# B&R Automation Studio project Prog_2
Automation Studio 4.5.2.102

## Configuration Config1

### Task classes (Cpu.sw)
```
Cyclic#1:
  Program <- Program.prg
Binaries: udbdef, TCData, ashwd, User, asfw, arconfig, sysconf, Role, ashwac, iomap, OpcUaMap
```

### Hardware
```
4PP065_0571_P74 : 4PP065.0571-P74 v1.1.2.0
  Connector IF5:
    ActivateDevice = 1
  ConfigurationID = Prog_2_Config1
  Simulation = 1
  ActivateOpcUa = 1
  OpcUa_SamplingTimer_Default = 1
  OpcUaInformationModels_PV_Version = 1
```

## Logical view

### Global.var
```iecst
VAR
	VP_At_Entry : BOOL;
	VP_At_Exit : BOOL;
	VP_Buffer_Conveyor : BOOL;
	VP_Entry_Conveyor : BOOL;
	VP_Item_Ready : BOOL;
	VP_Start_Button : BOOL;
	VP_Stop_Button : BOOL;
	VP_Dose_Button : BOOL;
END_VAR
```

### Program Logical/Program

#### Variables.var
```iecst
VAR
	RUN : BOOL;
	ENTRY_RUN : BOOL;
	DOSE : BOOL;
	RUN_TIME : UINT;
END_VAR
```

#### Main.c
```c
#include <bur/plctypes.h>

#ifdef _DEFAULT_INCLUDES
	#include <AsDefault.h>
#endif

void _INIT ProgramInit(void)
{

}

void _CYCLIC ProgramCyclic(void)
{
	if (VP_Start_Button) RUN = 1;
	if (!VP_Stop_Button) RUN = 0;

	if (RUN) {
		VP_Buffer_Conveyor = 1;

		if (!VP_Item_Ready) ENTRY_RUN = 1;
		if (VP_Dose_Button) DOSE = 1;

		if (!VP_At_Entry) {
			if (DOSE) ENTRY_RUN = 1;
			else ENTRY_RUN = 0;
		} else DOSE = 0;

		if (ENTRY_RUN) VP_Entry_Conveyor = 1;
		else VP_Entry_Conveyor = 0;

		if (!VP_Item_Ready || !VP_At_Entry) RUN_TIME = 0;
		if (RUN_TIME >= 350) {
			VP_Entry_Conveyor = 0;
			VP_Buffer_Conveyor = 0;
			RUN_TIME = 350;
		}

		RUN_TIME++;
	} else {
		VP_Entry_Conveyor = 0;
		VP_Buffer_Conveyor = 0;
	}
}

void _EXIT ProgramExit(void)
{

}
```
